(* CODESYS project FeedIceSequence.xml

Project tree, tasks and I/O mapping:
  function block FeedIceSequence [SFC]
*)

// FeedIceSequence
FUNCTION_BLOCK FeedIceSequence
// This function is for sequencing the ice feeding process. When triggered
// the output to feed ice is Set--then we wait for either the ice to be
// measured full by the ice full sensor, or a max feed time timeout.
// After the ice has been filled an additional top off time is allowed
// to run out. Then the fill ice output is Reset.

VAR_INPUT
	SFCInit: BOOL;
	Trigger: BOOL;
	IceFull: BOOL;
	MaxFeedTime: TIME;
	TopOffTime: TIME;
END_VAR
VAR_OUTPUT
	FillIce: BOOL;
	Complete: BOOL;
END_VAR
VAR
END_VAR

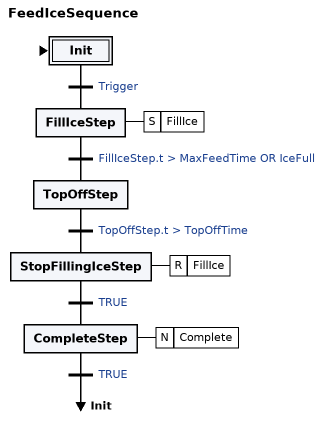
INITIAL_STEP Init:
END_STEP
TRANSITION FROM Init TO FillIceStep
    := Trigger;
END_TRANSITION
STEP FillIceStep:
    FillIce(S);
END_STEP
TRANSITION FROM FillIceStep TO TopOffStep
    := FillIceStep.t > MaxFeedTime OR IceFull;
END_TRANSITION
STEP TopOffStep:
END_STEP
TRANSITION FROM TopOffStep TO StopFillingIceStep
    := TopOffStep.t > TopOffTime;
END_TRANSITION
STEP StopFillingIceStep:
    FillIce(R);
END_STEP
TRANSITION FROM StopFillingIceStep TO CompleteStep
    := TRUE;
END_TRANSITION
STEP CompleteStep:
    Complete(N);
END_STEP
TRANSITION FROM CompleteStep TO Init
    := TRUE;
END_TRANSITION

END_FUNCTION_BLOCK
